SUBAPPLICATION mapping_DualOut_2_DO (* Subapplication Type *)
  (* Standard: 61499-2 *)
  (* Version 1.0, 2023-10-23, franz *)
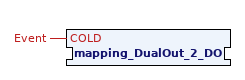
  EVENT_INPUT
    COLD;
  END_EVENT
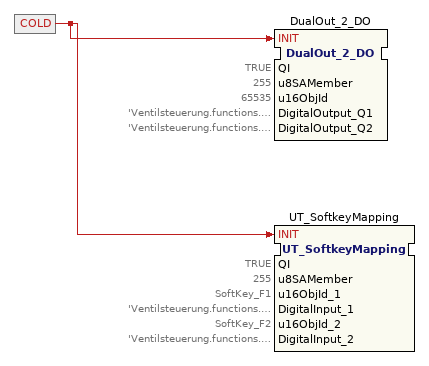
  FBS
    DualOut_2_DO : DualOut_2_DO(QI := TRUE, u8SAMember := 255, u16ObjId := 65535, DigitalOutput_Q1 := 'Ventilsteuerung.functions.DigitalOutput_Q1', DigitalOutput_Q2 := 'Ventilsteuerung.functions.DigitalOutput_Q2');
    UT_SoftkeyMapping : UT_SoftkeyMapping(QI := TRUE, u8SAMember := 255, u16ObjId_1 := SoftKey_F1, DigitalInput_1 := 'Ventilsteuerung.functions.SoftKey_F1', u16ObjId_2 := SoftKey_F2, DigitalInput_2 := 'Ventilsteuerung.functions.SoftKey_F2');
  END_FBS
  EVENT_CONNECTIONS
    COLD TO DualOut_2_DO.INIT;
    COLD TO UT_SoftkeyMapping.INIT;
  END_CONNECTIONS
END_SUBAPPLICATION
